FUNCTION "STREAM_CLEAR_1" : Void
{ S7_Optimized_Access := 'TRUE' }
VERSION : 0.1
   VAR_IN_OUT
      IN : "t_Stream";
   END_VAR


BEGIN
	"CLEAR_LS_1"(#IN.LString);
END_FUNCTION

